// TIA Portal V20 export
DATA_BLOCK "DB_HMI"   // DB4
{ S7_Optimized_Access := 'TRUE' }
// stored: MemoryReserve 100
   VAR
      Job_Mailbox : Array[0..3] of Word;
      Control_Screen : Word := 1;
      Alarm : Bool;
      Start : Bool;
      Change_Employee : Bool;
      Send_Recipe : Bool;
      Manual_Turn_On_Motor_Caroussel : Bool;
      Manual_Turn_On_Motor_Conveyor_Belt : Bool;
      Select_Test_Panel : SInt;
      Select_Motor_Speed : SInt := 1;
      Employee_Rework : String[6];
      Employee_Station_1 : String[6];
      Employee_Station_2 : String[6];
   END_VAR
   VAR RETAIN
      Admin_1 : String[6];
      Admin_2 : String[6];
      Admin_3 : String[6];
      Admin_4 : String[6];
      Admin_5 : String[6];
   END_VAR
   VAR
      Serial_Number : String[17];
      Electrical_Current : UInt;
      Electrical_Voltage : UInt;
      Electrical_Current_Result : String[10];
      Visual_Test_Result : String[10];
      Functional_Test_Result : String[10];
      Rework_Serial_Number : String[17];
      Rework_Electrical_Current : UInt;
      Rework_Electrical_Voltage : UInt;
      Rework_Electrical_Current_Result : String[10];
      Rework_Visual_Test_Result : String[10];
      Rework_Functional_Test_Result : String[10];
      Alarm_0 : Word;
      Alarm_1 : Word;
      Alarm_2 : Word;
   END_VAR
BEGIN
END_DATA_BLOCK
